(* IEC 61131-3 sources: plcassist-cli/packages/volt-cli/test/Volt.Ide.Twincat.Tests/fixtures/tc-workspace, 3 files *)

(* ---- FB_PackML_Unit.fb ---- *)
FUNCTION_BLOCK FB_PackML_Unit
VAR_INPUT
    xEmergencyStop  : BOOL;
    xSafetyOk       : BOOL;
    xPowerOn        : BOOL;
    xRemoteMode                 : BOOL;
    xMachineRunning : BOOL;

END_VAR
VAR_OUTPUT
    eState          : E_PackML_State;
    eMode           : E_PackML_Mode;
    ePrevState      : E_PackML_State;
    xStateChanged   : BOOL;
    xIdle           : BOOL;
    xExecute        : BOOL;
    xStopped        : BOOL;
    xComplete       : BOOL;
    xAborted        : BOOL;
    xHeld           : BOOL;
    xSuspended      : BOOL;
    nStatusWord     : WORD;
    nControlWord    : WORD;
    udiGoodCount    : UDINT;
    udiBadCount     : UDINT;
    udiTotalCount   : UDINT;
END_VAR
VAR
    fbModeManager   : FB_PackML_ModeManager;
    udiGoodCnt      : UDINT;
    udiBadCnt       : UDINT;
    xClearingDone   : BOOL;
    xResettingDone  : BOOL;
    xStartingDone   : BOOL;
    xCompletingDone : BOOL;
    xStoppingDone   : BOOL;
    xAbortingDone   : BOOL;
    xHoldingDone    : BOOL;
    xUnholdingDone  : BOOL;
    xSuspendingDone : BOOL;
    xUnsuspendingDone : BOOL;
    tonClearing     : TON;
    tonResetting    : TON;
    tonStarting     : TON;
    tonCompleting   : TON;
    tonStopping     : TON;
    tonAborting     : TON;
    tonHolding      : TON;
    tonUnholding    : TON;
    tonSuspending   : TON;
    tonUnsuspending : TON;
    tTmpTime        : TIME;
END_VAR

// ---------------------------------------------------------------------------
// Mode determination
// ---------------------------------------------------------------------------
IF NOT xPowerOn OR NOT xSafetyOk THEN
    eMode := E_PackML_Mode.eIDLE;
ELSIF xEmergencyStop THEN
    eMode := E_PackML_Mode.eIDLE;
ELSIF NOT xRemoteMode THEN
    eMode := E_PackML_Mode.eMANUAL;
ELSE
    eMode := E_PackML_Mode.ePRODUCTION;
END_IF

// ---------------------------------------------------------------------------
// Default timeout for step completion (override per state below)
// ---------------------------------------------------------------------------
tTmpTime := GVL_PackML.UNIT_STATE_TIMEOUT_DEFAULT;

// ---------------------------------------------------------------------------
// State-specific permissives & auto‑complete logic
// ---------------------------------------------------------------------------
CASE fbModeManager.eState OF

    E_PackML_State.eCLEARING:
        tTmpTime := T#5S;
        tonClearing(IN := TRUE, PT := tTmpTime);
        xClearingDone := tonClearing.Q;
        fbModeManager.xStateComplete := xClearingDone;

    E_PackML_State.eSTOPPED:
        tonClearing(IN := FALSE);
        tonResetting(IN := FALSE);
        fbModeManager.xStateComplete := FALSE;

    E_PackML_State.eRESETTING:
        tTmpTime := T#3S;
        tonResetting(IN := TRUE, PT := tTmpTime);
        xResettingDone := tonResetting.Q;
        fbModeManager.xStateComplete := xResettingDone;

    E_PackML_State.eIDLE:
        tonResetting(IN := FALSE);
        tonStarting(IN := FALSE);
        fbModeManager.xStateComplete := FALSE;

    E_PackML_State.eSTARTING:
        tTmpTime := T#3S;
        tonStarting(IN := TRUE, PT := tTmpTime);
        xStartingDone := tonStarting.Q;
        fbModeManager.xStateComplete := xStartingDone;

    E_PackML_State.eEXECUTE:
        tonStarting(IN := FALSE);
        tonCompleting(IN := FALSE);
        tonHolding(IN := FALSE);
        tonSuspending(IN := FALSE);
        fbModeManager.xStateComplete := FALSE;
        IF xMachineRunning THEN
            udiGoodCnt := udiGoodCnt + 1;
        END_IF

    E_PackML_State.eCOMPLETING:
        tTmpTime := T#3S;
        tonCompleting(IN := TRUE, PT := tTmpTime);
        xCompletingDone := tonCompleting.Q;
        fbModeManager.xStateComplete := xCompletingDone;

    E_PackML_State.eCOMPLETE:
        tonCompleting(IN := FALSE);
        fbModeManager.xStateComplete := FALSE;

    E_PackML_State.eHOLDING:
        tTmpTime := T#2S;
        tonHolding(IN := TRUE, PT := tTmpTime);
        xHoldingDone := tonHolding.Q;
        fbModeManager.xStateComplete := xHoldingDone;

    E_PackML_State.eHELD:
        tonHolding(IN := FALSE);
        tonUnholding(IN := FALSE);
        fbModeManager.xStateComplete := FALSE;

    E_PackML_State.eUNHOLDING:
        tTmpTime := T#2S;
        tonUnholding(IN := TRUE, PT := tTmpTime);
        xUnholdingDone := tonUnholding.Q;
        fbModeManager.xStateComplete := xUnholdingDone;

    E_PackML_State.eSUSPENDING:
        tTmpTime := T#2S;
        tonSuspending(IN := TRUE, PT := tTmpTime);
        xSuspendingDone := tonSuspending.Q;
        fbModeManager.xStateComplete := xSuspendingDone;

    E_PackML_State.eSUSPENDED:
        tonSuspending(IN := FALSE);
        tonUnsuspending(IN := FALSE);
        fbModeManager.xStateComplete := FALSE;

    E_PackML_State.eUNSUSPENDING:
        tTmpTime := T#2S;
        tonUnsuspending(IN := TRUE, PT := tTmpTime);
        xUnsuspendingDone := tonUnsuspending.Q;
        fbModeManager.xStateComplete := xUnsuspendingDone;

    E_PackML_State.eSTOPPING:
        tTmpTime := T#3S;
        tonStopping(IN := TRUE, PT := tTmpTime);
        xStoppingDone := tonStopping.Q;
        fbModeManager.xStateComplete := xStoppingDone;

    E_PackML_State.eABORTING:
        tTmpTime := T#2S;
        tonAborting(IN := TRUE, PT := tTmpTime);
        xAbortingDone := tonAborting.Q;
        fbModeManager.xStateComplete := xAbortingDone;

    E_PackML_State.eABORTED:
        tonAborting(IN := FALSE);
        fbModeManager.xStateComplete := FALSE;

END_CASE

// ---------------------------------------------------------------------------
// Call the mode manager
// ---------------------------------------------------------------------------
fbModeManager(
    xStart          := FALSE,
    xStop           := FALSE,
    xReset          := FALSE,
    xClear          := FALSE,
    xHold           := FALSE,
    xUnhold         := FALSE,
    xSuspend        := FALSE,
    xUnsuspend      := FALSE,
    xAbort          := xEmergencyStop OR NOT xSafetyOk,
    xStateComplete  := fbModeManager.xStateComplete
);

// ---------------------------------------------------------------------------
// Mirror outputs
// ---------------------------------------------------------------------------
eState        := fbModeManager.eState;
ePrevState    := fbModeManager.ePrevState;
xStateChanged := fbModeManager.xStateChanged;
xIdle         := fbModeManager.xIdle;
xExecute      := fbModeManager.xExecute;
xStopped      := fbModeManager.xStopped;
xComplete     := fbModeManager.xComplete;
xAborted      := fbModeManager.xAborted;
xHeld         := fbModeManager.xHeld;
xSuspended    := fbModeManager.xSuspended;

// ---------------------------------------------------------------------------
// Product counters
// ---------------------------------------------------------------------------
udiGoodCount  := udiGoodCnt;
udiBadCount   := udiBadCnt;
udiTotalCount := udiGoodCnt + udiBadCnt;

// ---------------------------------------------------------------------------
// OMAC / PackML Status Word (16-bit)
//   Bit 0–4  : State number (0–16)
//   Bit 5    : Suspended
//   Bit 6    : Held
//   Bit 7    : Complete
//   Bit 8    : Stopped
//   Bit 9    : Idle
//   Bit 10   : Execute
//   Bit 11   : Aborted
//   Bit 12   : Resetting
//   Bit 13   : Starting
//   Bit 14   : Alarming (reserved)
//   Bit 15   : Emergency / Fault
// ---------------------------------------------------------------------------
nStatusWord := USINT_TO_WORD(eState);
IF xSuspended  THEN nStatusWord.5  := TRUE; END_IF
IF xHeld       THEN nStatusWord.6  := TRUE; END_IF
IF xComplete   THEN nStatusWord.7  := TRUE; END_IF
IF xStopped    THEN nStatusWord.8  := TRUE; END_IF
IF xIdle       THEN nStatusWord.9  := TRUE; END_IF
IF xExecute    THEN nStatusWord.10 := TRUE; END_IF
IF xAborted    THEN nStatusWord.11 := TRUE; END_IF
IF eState = E_PackML_State.eRESETTING THEN nStatusWord.12 := TRUE; END_IF
IF eState = E_PackML_State.eSTARTING  THEN nStatusWord.13 := TRUE; END_IF
IF xEmergencyStop OR NOT xSafetyOk THEN nStatusWord.15 := TRUE; END_IF

// ---------------------------------------------------------------------------
// OMAC / PackML Control Word (16-bit) — for external HMI/PLC
//   Bit 0  : Start
//   Bit 1  : Stop
//   Bit 2  : Reset
//   Bit 3  : Clear
//   Bit 4  : Hold
//   Bit 5  : Unhold
//   Bit 6  : Suspend
//   Bit 7  : Unsuspend
//   Bit 8  : Abort
//   Bit 9  : Remote / Auto
//   Bit 10 : Reserved
//   Bit 11 : Reserved
//   Bit 12 : Reserved
//   Bit 13 : Reserved
//   Bit 14 : Reserved
//   Bit 15 : Reserved
// ---------------------------------------------------------------------------
nControlWord := 0;
IF xRemoteMode THEN
    nControlWord.9 := TRUE;
END_IF

END_FUNCTION_BLOCK

(* ---- FB_VltMembers.fb ---- *)
FUNCTION_BLOCK FB_VltMembers
VAR
	_level : INT;
END_VAR

_level := _level + 1;

METHOD PUBLIC Scale : INT
VAR_INPUT
	factor : INT;
END_VAR
VAR
	tmp : INT;
END_VAR

tmp := _level * factor;
Scale := tmp;
END_METHOD

PROPERTY PUBLIC Level : INT
GET
VAR
END_VAR
Level := _level;
END_GET
SET
VAR
END_VAR

_level := Level;
END_SET
END_PROPERTY

END_FUNCTION_BLOCK

(* ---- ladderLabel.prg ---- *)
PROGRAM ladderLabel
VAR
	coil: BOOL;
END_VAR

NETWORK 0 LD LABEL: testLabel
  coil := ;
END_NETWORK
NETWORK 1 LD LABEL: testLabe2
END_NETWORK

END_PROGRAM
